{attribute 'analysis' := '-33'}
TYPE RbtFanucUnloading_Array8Uint :
STRUCT
	_E: ARRAY [0..7] OF UINT;
END_STRUCT
END_TYPE

(* stored: Version 1.1.0.1
   DUT RbtFanucUnloading_Array8Uint: Id {5d5ed9d4-74a4-42d7-8e84-a85cd505c62b} *)
